{attribute addProperty BoxType "EP2001-1000-0016"}
{attribute addProperty Id "Group_0AT %Q*Group_5423B5073240Group_1AT %Q*Group_9433FC8D3240WcStateAT %I*WcState_28A8677510.1250InfoDataAT %I*InfoData_192954DE1620"}
{attribute addProperty CRC "3072731600"}
{attribute addProperty SizeInBites "81"}
{attribute addProperty SizeInBytes "10.125"}
TYPE EP2001_1F1194F3 :
STRUCT
	{attribute addProperty Name "Group_0"}
	Group_0 : Group_5423B507;
	{attribute addProperty Name "Group_1"}
	Group_1 : Group_9433FC8D;
	{attribute addProperty Name "WcState"}
	WcState : WcState_28A86775;
	{attribute addProperty Name "InfoData"}
	InfoData : InfoData_192954DE;
END_STRUCT
END_TYPE

(* stored: Version 1.2.0.0, ProductVersion 3.1.4024.9
   DUT EP2001_1F1194F3: Id {be2adeaa-b8b8-4e39-89db-328946efae45} *)
